FUNCTION CheckAlarm : BOOL
VAR_INPUT
	 pTank : POINTER TO ST_Tank;
END_VAR
VAR
END_VAR

IF pTank^.rtemperature >80 OR pTank^.rlevel > 90 THEN
	pTank^.bAlarm := TRUE;
	CheckAlarm := TRUE;
ELSE
		pTank^.bAlarm := FALSE;
		   CheckAlarm := FALSE;
END_IF

END_FUNCTION

(* stored: Version 1.1.0.1, ProductVersion 3.1.4024.16
   POU CheckAlarm: Id {e6ee15a6-c114-41f0-90a1-dfdd18b3a680}, SpecialFunc None *)
